FUNCTION_BLOCK Test_TStreamAdd_Read_REAL EXTENDS T_UnitTestBase
VAR
    Stream  : T_Stream(StreamLength := 2);
    ArgType : E_ArgTypeId := E_ArgTypeId.Type_REAL;
END_VAR

Stream.Init(2);

// add a REAL...
Stream.SetNextArgTypeId(ArgType);
Stream.Add_REAL(1.234567);

Stream.SetReadPosition(0);

// check next arg type is correct...
Assertion.AssertEquals_INT(Expected     := ArgType,
                           Actual       := Stream.GetNextArgTypeId(),
                           VariableName := 'Stream.GetNextArgTypeId()');

// check next value...	
Assertion.AssertEquals_REAL(Expected     := 1.234567,
                            Actual       := Stream.Read_REAL(),
                            Delta        := 0.000001,
                            VariableName := 'Stream.Read_REAL()');

// check we are at the end of the stream..							
Assertion.AssertEquals_UDINT(Expected     := Stream.StreamLength,
                             Actual       := Stream.ReadPosition,
                             VariableName := 'Stream.ReadPosition');

TestFinished();

END_FUNCTION_BLOCK

(* stored: Version 1.1.0.1, ProductVersion 3.1.4024.9
   POU Test_TStreamAdd_Read_REAL: Id {f6f24f4f-449f-4d4b-9188-09f3d21a95c8}, SpecialFunc None *)
